{attribute 'qualified_only'}
VAR_GLOBAL

END_VAR

(* stored: Version 1.1.0.1, ProductVersion 3.1.4024.12
   GVL GVL_SL2K4: Id {fc41bd45-f004-43ad-8266-dcc2d3ff2d2e} *)
